RoboDK station: BottleDetection_YOLOv8.rdk

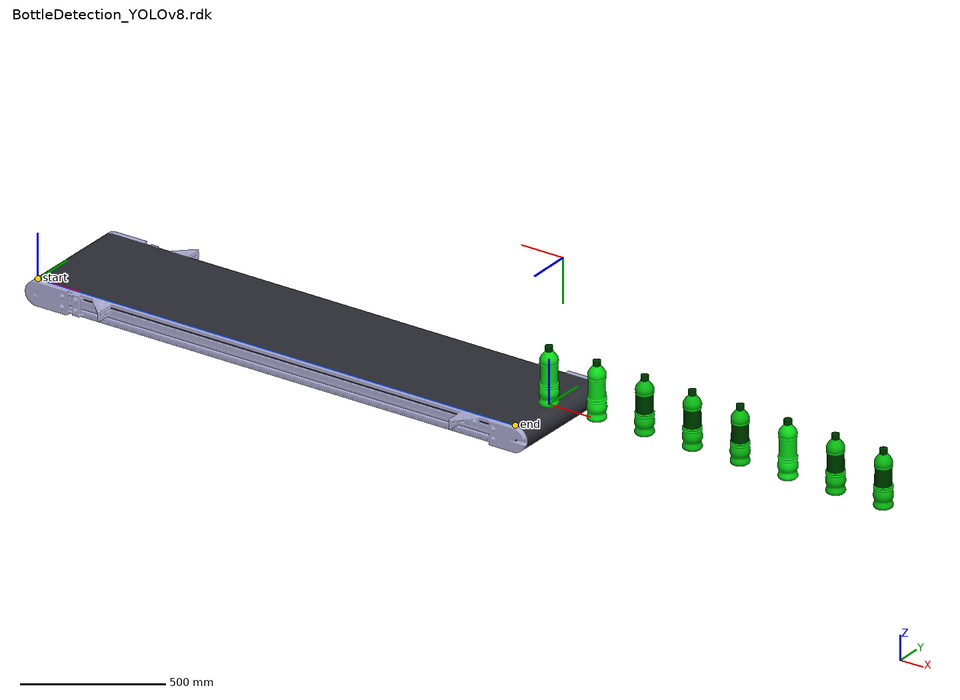
[picture v0: the station drawn from its stored meshes, robots at their saved joint values, targets as dots, program paths as lines]
Station BottleDetection_YOLOv8 (saved by RoboDK 5.6.8). Poses are relative to the parent item; angles as X-Y-Z fixed-axis rotations.
  - Python program box (listed below)
  - frame Camera at (1500, 1000, 100) mm, rotated rx -90 ry 0 rz 180 deg
    - camera camera
  - program Prog1 (3 instructions, listed below)
  - frame Conveyor Belt (2m) Base at (0, 0, 0) mm
    - robot Conveyor Belt (2m): 1 axes
        modified DH rows (alpha deg, a mm, theta deg, d mm): 0, 0, 0, 0 linear
        base shift (0, 0, 0) mm, rotated rx 0 ry 90 rz 0 deg
        joint limits [-500000] to [500000]; home [0]; saved at [2000]
      - frame Frame 2 at (0, 200, 0) mm
        - object Bottle (Plain) at (0, 0, 0) mm, size 71.4 x 71.4 x 225.2 mm, geometry from Bottle-Plain.sld
        - object Bottle (Plain) at (0, 0, 0) mm, size 71.4 x 71.4 x 225.2 mm, geometry from Bottle-Plain.sld
        - object Bottle (Label) at (0, 0, 0) mm, size 71.4 x 71.4 x 225.2 mm, geometry from Bottle-Label (1).sld
        - object Bottle (Label) at (0, 0, 0) mm, size 71.4 x 71.4 x 225.2 mm, geometry from Bottle-Label (1).sld
        - object Bottle (Plain) at (0, 0, 0) mm, size 71.4 x 71.4 x 225.2 mm, geometry from Bottle-Plain.sld
        - object Bottle (Label) at (0, 0, 0) mm, size 71.4 x 71.4 x 225.2 mm, geometry from Bottle-Label (1).sld
        - object Bottle (Label) at (0, 0, 0) mm, size 71.4 x 71.4 x 225.2 mm, geometry from Bottle-Label (1).sld
        - object Bottle (Label) at (0, 0, 0) mm, size 71.4 x 71.4 x 225.2 mm, geometry from Bottle-Label (1).sld
    - target start (Cartesian target) at (0, 0, 0) mm; joints [0] of Conveyor Belt (2m)
    - target end (Cartesian target) at (2000, 0, 0) mm; joints [2000] of Conveyor Belt (2m)
  - Python program Prog2 (listed below)
  - Python program Ultra (listed below)
  - Python program Ultrabox (listed below)

--- Python program box ---
from robodk.robolink import *  # RoboDK API
from roboflow import Roboflow
import cv2 as cv
import numpy as np
import json

#----------------------------------
# Settings
PROCESS_COUNT = -1  # How many frames to process before exiting. -1 means indefinitely.

CAM_NAME = "camera"  # Change the camera name here to match your camera name

DISPLAY_SETTINGS = True
WDW_NAME_PARAMS = 'RoboDK - Blob detection parameters'

DISPLAY_RESULT = True
WDW_NAME_RESULTS = 'RoboDK - Blob detections'

#----------------------------------
# Get the simulated camera from RoboDK
RDK = Robolink()

cam_item = RDK.Item(CAM_NAME, ITEM_TYPE_CAMERA)
if not cam_item.Valid():
    raise Exception("Camera not found! %s" % CAM_NAME)
cam_item.setParam('Open', 1)  # Force the camera view to open

# Initialize the Roboflow API
rf = Roboflow(api_key="GYx3tvb9zCC6sFvjakIJ")
project = rf.workspace("malaria-1ml5u").project("bottle-lxw4g")
model = project.version(2).model

#----------------------------------------------
# Set up the detector with default parameters.
# Default parameters extract dark circular blobs.
params = cv.SimpleBlobDetector_Params()
detector = cv.SimpleBlobDetector_create(params)

#----------------------------------------------
# Set up sliders for parameters, using OpenCV's trackbars
if DISPLAY_SETTINGS:
    # Your code for setting up sliders goes here

#----------------------------------------------
# Create a resizable result window
   if DISPLAY_RESULT:
       cv.namedWindow(WDW_NAME_RESULTS)

#----------------------------------------------
# Start processing camera frames
count = 0
while count < PROCESS_COUNT or PROCESS_COUNT < 0:
    print("=============================================")
    print("Processing image %i" % count)
    count += 1

    # Get the image from RoboDK
    bytes_img = RDK.Cam2D_Snapshot("", cam_item)
    if bytes_img == b'':
        raise Exception("Failed to capture image from camera.")
    nparr = np.frombuffer(bytes_img, np.uint8)
    frame = cv.imdecode(nparr, cv.IMREAD_COLOR)
    if frame is None or frame.shape == ():
        raise Exception("Failed to decode image.")

    # Perform blob detection
    keypoints = detector.detect(frame)

    # Perform object detection using Roboflow API
    prediction_response = model.predict(frame, confidence=40, overlap=30).json()

    # Extract class and bounding box coordinates
    for prediction in prediction_response['predictions']:
        class_name = prediction['class']
        x, y, width, height = prediction['x'], prediction['y'], prediction['width'], prediction['height']

        # Draw bounding boxes around the detected objects
        cv.rectangle(frame, (int(x), int(y)), (int(x + width), int(y + height)), (255, 0, 0), 2)
        cv.putText(frame, class_name, (int(x), int(y) - 5), cv.FONT_HERSHEY_SIMPLEX, 0.5, (255, 255, 0), 2)

    # Display the detection results
    if DISPLAY_RESULT:
        # Draw detected blobs and their id
        img_matches = cv.drawKeypoints(frame, keypoints, None, (0, 255, 0), cv.DRAW_MATCHES_FLAGS_DRAW_RICH_KEYPOINTS)
        i = 0
        for keypoint in keypoints:
            x, y = keypoint.pt
            cv.putText(img_matches, str(i), (int(x), int(y)), cv.FONT_HERSHEY_SIMPLEX, 1, (0, 255, 0), 1, cv.LINE_AA)
            i += 1

        # Resize the image
        img_matches = cv.resize(img_matches, (int(img_matches.shape[1] * .75), int(img_matches.shape[0] * .75)))

        cv.imshow(WDW_NAME_RESULTS, img_matches)
        key = cv.waitKey(500)
        if key == 27:
            break  # User pressed ESC, exit
        if cv.getWindowProperty(WDW_NAME_RESULTS, cv.WND_PROP_VISIBLE) < 1:
            break  # User closed the window, exit

cv.destroyAllWindows()

--- program Prog1 (robot Conveyor Belt (2m)) ---
  Set Ref.: Conveyor Belt (2m) Base
  MoveJ (start)
  MoveJ (end)

--- Python program Prog2 ---
from robodk.robolink import *  # RoboDK API
from roboflow import Roboflow
import cv2 as cv
import numpy as np
import json

#----------------------------------
# Settings
PROCESS_COUNT = -1  # How many frames to process before exiting. -1 means indefinitely.

CAM_NAME = "camera"  # Change the camera name here to match your camera name

DISPLAY_SETTINGS = True
WDW_NAME_PARAMS = 'RoboDK - Blob detection parameters'

DISPLAY_RESULT = True
WDW_NAME_RESULTS = 'RoboDK - Blob detections'

#----------------------------------
# Get the simulated camera from RoboDK
RDK = Robolink()

cam_item = RDK.Item(CAM_NAME, ITEM_TYPE_CAMERA)
if not cam_item.Valid():
    raise Exception("Camera not found! %s" % CAM_NAME)
cam_item.setParam('Open', 1)  # Force the camera view to open

# Initialize the Roboflow API
rf = Roboflow(api_key="GYx3tvb9zCC6sFvjakIJ")
project = rf.workspace("malaria-1ml5u").project("bottle-lxw4g")
model = project.version(2).model

#----------------------------------------------
# Set up the detector with default parameters.
# Default parameters extract dark circular blobs.
params = cv.SimpleBlobDetector_Params()
detector = cv.SimpleBlobDetector_create(params)

#----------------------------------------------
# Set up sliders for parameters, using OpenCV's trackbars
if DISPLAY_SETTINGS:
    # Your code for setting up sliders goes here

#----------------------------------------------
# Create a resizable result window
  if DISPLAY_RESULT:
      cv.namedWindow(WDW_NAME_RESULTS)

#----------------------------------------------
# Start processing camera frames
count = 0
while count < PROCESS_COUNT or PROCESS_COUNT < 0:
    print("=============================================")
    print("Processing image %i" % count)
    count += 1

    # Get the image from RoboDK
    bytes_img = RDK.Cam2D_Snapshot("", cam_item)
    if bytes_img == b'':
        raise Exception("Failed to capture image from camera.")
    nparr = np.frombuffer(bytes_img, np.uint8)
    img = cv.imdecode(nparr, cv.IMREAD_UNCHANGED)
    if img is None or img.shape == ():
        raise Exception("Failed to decode image.")

    # Perform blob detection
    keypoints = detector.detect(img)

    # Perform object detection using Roboflow API
    prediction_response = model.predict(img, confidence=40, overlap=30).json()

    # Extract class and x, y values
    predictions = prediction_response['predictions']

    # Process inference results
    for prediction in predictions:
        class_name = prediction['class']
        x, y, width, height = prediction['x'], prediction['y'], prediction['width'], prediction['height']

        print(f"Class: {class_name}, X: {x}, Y: {y}, Width: {width}, Height: {height}")

    # Display the detection results
    if DISPLAY_RESULT:
        # Draw detected blobs and their id
        img_matches = cv.drawKeypoints(img, keypoints, None, (0, 255, 0), cv.DRAW_MATCHES_FLAGS_DRAW_RICH_KEYPOINTS)
        i = 0
        for keypoint in keypoints:
            x, y = keypoint.pt
            cv.putText(img_matches, str(i), (int(x), int(y)), cv.FONT_HERSHEY_SIMPLEX, 1, (0, 255, 0), 1, cv.LINE_AA)
            i += 1

        # Resize the image
        img_matches = cv.resize(img_matches, (int(img_matches.shape[1] * .75), int(img_matches.shape[0] * .75)))

        cv.imshow(WDW_NAME_RESULTS, img_matches)
        key = cv.waitKey(500)
        if key == 27:
            break  # User pressed ESC, exit
        if cv.getWindowProperty(WDW_NAME_RESULTS, cv.WND_PROP_VISIBLE) < 1:
            break  # User closed the window, exit

cv.destroyAllWindows()

--- Python program Ultra ---
from robodk.robolink import *  # RoboDK API
from ultralytics import YOLO
import cv2 as cv
import numpy as np

#----------------------------------
# Settings
PROCESS_COUNT = -1  # How many frames to process before exiting. -1 means indefinitely.

CAM_NAME = "camera"  # Change the camera name here to match your camera name

DISPLAY_SETTINGS = True
WDW_NAME_PARAMS = 'RoboDK - Blob detection parameters'

DISPLAY_RESULT = True
WDW_NAME_RESULTS = 'RoboDK - Blob detections'

#----------------------------------
# Get the simulated camera from RoboDK
RDK = Robolink()

cam_item = RDK.Item(CAM_NAME, ITEM_TYPE_CAMERA)
if not cam_item.Valid():
    raise Exception("Camera not found! %s" % CAM_NAME)
cam_item.setParam('Open', 1)  # Force the camera view to open

# Load a pretrained YOLOv5 model
model = YOLO('C:/Users/joelb/OneDrive/Documents/RoboDK/bottle.pt')

#----------------------------------------------
# Set up the detector with default parameters.
# Default parameters extract dark circular blobs.
params = cv.SimpleBlobDetector_Params()
detector = cv.SimpleBlobDetector_create(params)

#----------------------------------------------
# Set up sliders for parameters, using OpenCV's trackbars
if DISPLAY_SETTINGS:
    # Your code for setting up sliders goes here

#----------------------------------------------
# Create a resizable result window
   if DISPLAY_RESULT:
        cv.namedWindow(WDW_NAME_RESULTS)

#----------------------------------------------
# Start processing camera frames
count = 0
while count < PROCESS_COUNT or PROCESS_COUNT < 0:
    print("=============================================")
    print("Processing image %i" % count)
    count += 1

    # Get the image from RoboDK
    bytes_img = RDK.Cam2D_Snapshot("", cam_item)
    if bytes_img == b'':
        raise Exception("Failed to capture image from camera.")
    nparr = np.frombuffer(bytes_img, np.uint8)
    img = cv.imdecode(nparr, cv.IMREAD_UNCHANGED)
    if img is None or img.shape == ():
        raise Exception("Failed to decode image.")

    # Perform blob detection
    keypoints = detector.detect(img)

    # Perform object detection using YOLOv5 model
    results = model(img)  # list of Results objects

    # Display the detection results
    if DISPLAY_RESULT:
        # Resize the image
        img = cv.resize(img, (int(img.shape[1] * .75), int(img.shape[0] * .75)))

        cv.imshow(WDW_NAME_RESULTS, img)
        key = cv.waitKey(500)
        if key == 27:
            break  # User pressed ESC, exit
        if cv.getWindowProperty(WDW_NAME_RESULTS, cv.WND_PROP_VISIBLE) < 1:
            break  # User closed the window, exit

cv.destroyAllWindows()

--- Python program Ultrabox ---
from robodk.robolink import *  # RoboDK API
from ultralytics import YOLO
import cv2
import numpy as np
import os
import math
from robolink import import_install

#----------------------------------
# Settings
PROCESS_COUNT = -1  # How many frames to process before exiting. -1 means indefinitely.
OUTPUT_DIR = "output_images"  # Directory to save the inference results

CAM_NAME = "camera"  # Change the camera name here to match your camera name

#DISPLAY_SETTINGS = True
WDW_NAME_PARAMS = 'RoboDK - Blob detection parameters'

DISPLAY_RESULT = True
WDW_NAME_RESULTS = 'RoboDK - Blob detections'

# Create the output directory if it doesn't exist
if not os.path.exists(OUTPUT_DIR):
    os.makedirs(OUTPUT_DIR)

#----------------------------------
# Get the simulated camera from RoboDK
RDK = Robolink()

cam_item = RDK.Item(CAM_NAME, ITEM_TYPE_CAMERA)
if not cam_item.Valid():
    raise Exception("Camera not found! %s" % CAM_NAME)
cam_item.setParam('Open', 1)  # Force the camera view to open

# Load a pretrained YOLOv5 model
model = YOLO('C:/Users/joelb/OneDrive/Documents/RoboDK/bottle.pt')
classnames = ['label','no_label']

#----------------------------------------------
# Set up the detector with default parameters.
# Default parameters extract dark circular blobs.
params = cv2.SimpleBlobDetector_Params()
detector = cv2.SimpleBlobDetector_create(params)

#----------------------------------------------
# Start processing camera frames
count = 0
while count < PROCESS_COUNT or PROCESS_COUNT < 0:
    print("=============================================")
    print("Processing image %i" % count)
    count += 1

    # Get the image from RoboDK
    bytes_img = RDK.Cam2D_Snapshot("", cam_item)
    if bytes_img == b'':
        raise Exception("Failed to capture image from camera.")
    nparr = np.frombuffer(bytes_img, np.uint8)
    frame = cv2.imdecode(nparr, cv2.IMREAD_COLOR)  # Ensure image has 3 channels (RGB)
    if frame is None or frame.shape[2] != 3:
        raise Exception("Failed to decode image or incorrect number of channels.")

    # Perform blob detection
    keypoints = detector.detect(frame)

    # Perform object detection using YOLOv5 model
    results = model(frame)  # list of Results objects

    # Draw bounding boxes around the detected objects
    for info in results:
        parameters = info.boxes
        for box in parameters:
            x1, y1, x2, y2 = box.xyxy[0]
            x1, y1, x2, y2 = int(x1), int(y1), int(x2), int(y2)
            confidence = box.conf[0]
            class_detect = box.cls[0]
            class_detect = int(class_detect)
            class_detect = classnames[class_detect]
            conf = math.ceil(confidence * 100)
            cv2.rectangle(frame, (x1, y1), (x2, y2), (0, 255, 0), 2)
            cv2.putText(frame, f'{class_detect}', (x1 + 8, y1 - 12), cv2.FONT_HERSHEY_DUPLEX, 1, (255,165,0), 1, cv2.LINE_AA)

    # Save the inference result
    output_path = os.path.join(OUTPUT_DIR, f"C:/RoboDK/inference/result_{count}.jpg")
    cv2.imwrite(output_path, frame)
    print(f"Inference result saved to: {output_path}")

    # Display the detection results
    if DISPLAY_RESULT:
        # Resize the image
        frame = cv2.resize(frame, (int(frame.shape[1] * .75), int(frame.shape[0] * .75)))

        cv2.imshow(WDW_NAME_RESULTS, frame)
        key = cv2.waitKey(500)
        if key == 27:
            break  # User pressed ESC, exit
        if cv2.getWindowProperty(WDW_NAME_RESULTS, cv2.WND_PROP_VISIBLE) < 1:
            break  # User closed the window, exit

cv2.destroyAllWindows()
